FUNCTION_BLOCK TcaSegmentDoor EXTENDS TcoComponent

VAR_INPUT
	ref : REFERENCE TO TcaSegmentDoorRef;
END_VAR

VAR
	_status : TcaSegmentDoorStatus;
	_config : TcaSegmentDoorConfig;
	_service : TcaSegmentDoorService;
	
	//Tasks
	_closeTask : TcoCore.TcoTask(THIS^);
	_openTask : TcoCore.TcoTask(THIS^);
	_initTask : TcoCore.TcoTask(THIS^);
	
	_EnableAxis : BOOL := TRUE;
	_EnableAxisSafe : BOOL;
	
	// Components
	_vertikalAxis : TcoDriveSimple(THIS^);	
	_latchLeft : TcoDriveSimple(THIS^);
	_latchRight : TcoDriveSimple(This^);

END_VAR

IF NOT __ISVALIDREF(ref)  THEN
    Messenger.Post('<#Invalid reference signal #>', TcoCore.eMessageCategory.ProgrammingError);
    RETURN;
END_IF

// Axis
_EnableAxisSafe := _EnableAxis; //AND ref.tsSS1;
_vertikalAxis(inCalibrationCam:= ref.ReferenceSensor, inEnable:=  _EnableAxisSafe , inEnableNegative:= _EnableAxisSafe, inEnablePositive:= _EnableAxisSafe, inoAxisRef:= ref.VertikalAxis);
_latchLeft( inEnable:= _EnableAxisSafe, inEnableNegative:= _EnableAxisSafe, inEnablePositive:= _EnableAxisSafe, inoAxisRef:= ref.LatchLeft);
_latchRight( inEnable:= _EnableAxisSafe, inEnableNegative:= _EnableAxisSafe, inEnablePositive:= _EnableAxisSafe, inoAxisRef:= ref.LatchRight);

METHOD Close : ITcoTaskStatus
VAR_INPUT
END_VAR
_closeTask.Restore();
Close := _closeTask.Invoke();
END_METHOD

PROPERTY CloseTask : TcoCore.ITcoTask
GET
CloseTask := _CloseTask;
END_GET
END_PROPERTY

PROPERTY Config : REFERENCE TO TcaSegmentDoorConfig
GET
Config Ref= _config;
END_GET
SET
_config := Config;
END_SET
END_PROPERTY

METHOD Init : ITcoTaskStatus
VAR_INPUT
END_VAR
_closeTask.Restore();
Init := _closeTask.Invoke();
END_METHOD

PROPERTY InitTask : TcoCore.ITcoTask
GET
InitTask := _InitTask;
END_GET
END_PROPERTY

METHOD Open : ITcoTaskStatus
VAR_INPUT
END_VAR
_openTask.Restore();
Open := _openTask.Invoke();
END_METHOD

PROPERTY OpenTask : TcoCore.ITcoTask
GET
OpenTask := _OpenTask;
END_GET
END_PROPERTY

{warning 'Methodenimplementierung hinzufügen'}
METHOD Restore : TcoCore.ITcoRestorable
END_METHOD

{warning 'Methodenimplementierung hinzufügen'}
(*~
	<docu>
		<summary>
		    Custom service (manual, maintenance) logic.
			This method must be implemented in derived class.
		</summary>			
	</docu>	
~*)
METHOD PROTECTED ServiceMode
END_METHOD

PROPERTY Status : REFERENCE TO TcaSegmentDoorStatus
GET
Status REF= _status;
END_GET
END_PROPERTY

END_FUNCTION_BLOCK

(* stored: Version 1.1.0.1
   POU TcaSegmentDoor: Id {ad4e5a73-bf23-4c54-b7b1-393428a1c398}, SpecialFunc None
   Folder Functions: Id {aa5400d1-3e83-4e87-8cbe-7fdaf6dd4d10}
   Folder Operations: Id {0337acaf-bb1e-4ccc-8f29-a9d1ea5cf9cf}
   Folder States: Id {6e7f2e8f-37a8-4f05-a8c3-d2e8d57a07dd}
   Folder Tasks: Id {838c9210-3ca4-442a-a07e-a6d989e5a17d}
   Method Close: Id {da8c0a98-2224-40bd-9fb9-d56e5af75aab}
   Property CloseTask: Id {fdcb56f2-347b-4635-b675-1976c0f30f02}
   Get Get: Id {581f66b8-0280-4f39-81d0-e63d63281ad3}
   Property Config: Id {c68b7b98-0a10-4d8d-8e62-47f2197e8467}
   Get Get: Id {0903fc32-f9cf-4b6b-aa89-f6457dbcad7d}
   Set Set: Id {c6353d11-4afa-4ff3-9eee-8a5ebd46d5f8}
   Method Init: Id {a0790239-fb81-4898-923e-8f66a94daf78}
   Property InitTask: Id {4d213dad-e52e-48a2-a9ec-2162ee141fe6}
   Get Get: Id {e0361ccd-174f-426d-8378-68b4d0f0a754}
   Method Open: Id {43b934e2-9d63-4d46-86fe-8299edf7fc0c}
   Property OpenTask: Id {c78f4c29-2ad9-4500-854e-86d65951471d}
   Get Get: Id {d9d5923e-4f9a-411f-b7ef-f21be615cc55}
   Method Restore: Id {d83d557c-7a15-4d4d-9b23-bc93b0b1c613}
   Method ServiceMode: Id {364f241a-3f02-4572-bd41-45a4ab035d33}
   Property Status: Id {7c350292-0925-4da3-830a-845fdcb91274}
   Get Get: Id {c1b1edc5-850b-4b60-a166-968539086957} *)
